// TwinCAT 3 PLC project Test_OnlineChange
// ProgramVersion: 3.1.4026.22
// libraries:
//   Tc2_Standard, * (Beckhoff Automation GmbH)
//   Tc2_System, * (Beckhoff Automation GmbH)
//   Tc3_JsonXml, * (Beckhoff Automation GmbH)
//   Stage, * (_)
// project tree:
//   DUTs/ T_OnlineChangeTestCheck.TcDUT, T_OnlineChangeTestChecks.TcDUT, T_OnlineChangeTestEntity.TcDUT, T_OnlineChangeTestExecute.TcDUT, T_OnlineChangeTestReport.TcDUT, T_OnlineChangeTestRuntime.TcDUT, T_OnlineChangeTestStage.TcDUT, T_OnlineChangeTestWorker.TcDUT
//   GVLs/ GVL_OnlineChangeTest.TcGVL
//   POUs/ FB_OnlineChangeProbe.TcPOU, FB_OnlineChangeDefineReset.TcPOU, FB_OnlineChangeJsonReport.TcPOU, FB_OnlineChangeMovePadding.TcPOU, FB_OnlineChangeStageMarker.TcPOU, FB_FastThreadConfig.TcPOU, FB_TestExecute.TcPOU, FB_TestJob.TcPOU, MAIN.TcPOU
//   / PlcTask.TcTTO
// (motion and I/O tree: see PLC project stage)
// real-time tasks:
//   TASK Example: cycle T#10ms, priority 20, ADS port 350
//   TASK Test: cycle T#10ms, priority 21, ADS port 351
//   TASK VISU_TASK: cycle T#200000us, priority 30, ADS port 352
//   TASK PlcTask: cycle T#10ms, priority 22, ADS port 353
//   TASK PlcTask1: cycle T#10ms, priority 23, ADS port 354
//   TASK PlcTask2: cycle T#10ms, priority 24, ADS port 355

CONFIGURATION Test_OnlineChange
    RESOURCE PLC ON TwinCAT3
        TASK PlcTask(INTERVAL := T#10ms, PRIORITY := 24);
        PROGRAM MAIN WITH PlcTask : MAIN;
    END_RESOURCE
END_CONFIGURATION

// ---- DUTs/T_OnlineChangeTestCheck.TcDUT
TYPE T_OnlineChangeTestCheck :
STRUCT
	bRequired: BOOL;
	bPassed: BOOL;
END_STRUCT
END_TYPE

// ---- DUTs/T_OnlineChangeTestChecks.TcDUT
TYPE T_OnlineChangeTestChecks :
STRUCT
	NoPanic: T_OnlineChangeTestCheck;
	StageSelected: T_OnlineChangeTestCheck;
	StableCallback: T_OnlineChangeTestCheck;
	NoChangeFlags: T_OnlineChangeTestCheck;
	AddDeleteFlags: T_OnlineChangeTestCheck;
	CreatedInit: T_OnlineChangeTestCheck;
	CreatedCallback: T_OnlineChangeTestCheck;
	RepairWarn: T_OnlineChangeTestCheck;
	ActiveJobRunning: T_OnlineChangeTestCheck;
	IdleJobStarted: T_OnlineChangeTestCheck;
	MovedCallback: T_OnlineChangeTestCheck;
	MovedExecuteRunning: T_OnlineChangeTestCheck;
	MovedJobRunning: T_OnlineChangeTestCheck;
END_STRUCT
END_TYPE

// ---- DUTs/T_OnlineChangeTestEntity.TcDUT
TYPE T_OnlineChangeTestEntity :
STRUCT
	nStableInit: UDINT;
	nRemovedInit: UDINT;
	nCreatedInit: UDINT;

	nStableOnlineChange: UDINT;
	bStableLastEntityCreated: BOOL;
	bStableLastEntityDeleted: BOOL;

	nCreatedOnlineChange: UDINT;
	bCreatedLastEntityCreated: BOOL;
	bCreatedLastEntityDeleted: BOOL;

	nMovedInit: UDINT;
	nMovedOnlineChange: UDINT;
	bMovedLastEntityCreated: BOOL;
	bMovedLastEntityDeleted: BOOL;
END_STRUCT
END_TYPE

// ---- DUTs/T_OnlineChangeTestExecute.TcDUT
TYPE T_OnlineChangeTestExecute :
STRUCT
	nMainCycles: UDINT;
	nThreadedCycles: UDINT;
	nMovedCycles: UDINT;
END_STRUCT
END_TYPE

// ---- DUTs/T_OnlineChangeTestReport.TcDUT
TYPE T_OnlineChangeTestReport :
STRUCT
	bAllRequiredPassed: BOOL;
	bRequiredFailure: BOOL;
	bJsonReady: BOOL;
	bJsonCopyOk: BOOL;
	nJsonLength: UDINT;
	sJson: STRING(2048);
END_STRUCT
END_TYPE

// ---- DUTs/T_OnlineChangeTestRuntime.TcDUT
TYPE T_OnlineChangeTestRuntime :
STRUCT
	nMainCycles: UDINT;
	nTotalPanic: UDINT;
	nTotalWarn: UDINT;
END_STRUCT
END_TYPE

// ---- DUTs/T_OnlineChangeTestStage.TcDUT
TYPE T_OnlineChangeTestStage :
STRUCT
	sName: STRING(80);
	nId: UINT;
	iConfiguredFastThread: Stage.I_Thread;
	bFastThreadConfigured: BOOL;
END_STRUCT
END_TYPE

// ---- DUTs/T_OnlineChangeTestWorker.TcDUT
TYPE T_OnlineChangeTestWorker :
STRUCT
	nActiveInit: UDINT;
	nActiveExecute: UDINT;
	nActiveExit: UDINT;
	nIdleInit: UDINT;
	nIdleExecute: UDINT;
	nIdleExit: UDINT;
	nMovedInit: UDINT;
	nMovedExecute: UDINT;
	nMovedExit: UDINT;

	nActiveStartOk: UDINT;
	nActiveStartNone: UDINT;
	nActiveStartError: UDINT;
	nIdleStartOk: UDINT;
	nIdleStartNone: UDINT;
	nIdleStartError: UDINT;
	nMovedStartOk: UDINT;
	nMovedStartNone: UDINT;
	nMovedStartError: UDINT;

	bActiveStartRequested: BOOL;
	bIdleStartRequested: BOOL;
	bMovedStartRequested: BOOL;

	eActiveState: Stage.JobState;
	eIdleState: Stage.JobState;
	eMovedState: Stage.JobState;
END_STRUCT
END_TYPE

// ---- GVLs/GVL_OnlineChangeTest.TcGVL
{attribute 'qualified_only'}
VAR_GLOBAL
	StageState: T_OnlineChangeTestStage;
	Runtime: T_OnlineChangeTestRuntime;
	Entity: T_OnlineChangeTestEntity;
	Execute: T_OnlineChangeTestExecute;
	Worker: T_OnlineChangeTestWorker;
	Checks: T_OnlineChangeTestChecks;
	Report: T_OnlineChangeTestReport;
END_VAR

// ---- POUs/MAIN.TcPOU
// TEST_OC_STAGE values:
// 'INIT' = init baseline
// 'NO_CHANGE' = same-shape online change
// 'REMOVE_THREAD' = remove fast thread
// 'ADD_DELETE_ENTITY' = add/delete entity
// 'MOVE_MEMORY' = force stable instances to move inside program memory
PROGRAM MAIN
{define TEST_OC_STAGE 'MOVE_MEMORY'}
VAR
	fbDefineReset: FB_OnlineChangeDefineReset;
	fbJsonReport: FB_OnlineChangeJsonReport;

	fbStableProbe: FB_OnlineChangeProbe(1);
	fbMainExecute: FB_TestExecute(1);
	fbThreadedExecute: FB_TestExecute(2);
	fbActiveJob: FB_TestJob(1);
	fbIdleJob: FB_TestJob(2);

{IF hasvalue(TEST_OC_STAGE, 'INIT')}
	fbStageInit: FB_OnlineChangeStageMarker(1);
	fbFastThread: Stage.Thread;
	fbFastConfig: FB_FastThreadConfig(fbFastThread);
	fbRemovedProbe: FB_OnlineChangeProbe(2);
{END_IF}
{IF hasvalue(TEST_OC_STAGE, 'NO_CHANGE')}
	fbStageNoChange: FB_OnlineChangeStageMarker(2);
	fbFastThread: Stage.Thread;
	fbFastConfig: FB_FastThreadConfig(fbFastThread);
	fbRemovedProbe: FB_OnlineChangeProbe(2);
{END_IF}
{IF hasvalue(TEST_OC_STAGE, 'REMOVE_THREAD')}
	fbStageRemoveThread: FB_OnlineChangeStageMarker(3);
	fbRemovedProbe: FB_OnlineChangeProbe(2);
{END_IF}
{IF hasvalue(TEST_OC_STAGE, 'ADD_DELETE_ENTITY')}
	fbStageAddDeleteEntity: FB_OnlineChangeStageMarker(4);
	fbCreatedProbe: FB_OnlineChangeProbe(3);
{END_IF}
{IF hasvalue(TEST_OC_STAGE, 'MOVE_MEMORY')}
	fbStageMoveMemory: FB_OnlineChangeStageMarker(5);
	fbFastThread: Stage.Thread;
	fbFastConfig: FB_FastThreadConfig(fbFastThread);
	fbRemovedProbe: FB_OnlineChangeProbe(2);
{END_IF}

{IF hasvalue(TEST_OC_STAGE, 'INIT')}
	fbMovePadInit: FB_OnlineChangeMovePadding;
{END_IF}
{IF hasvalue(TEST_OC_STAGE, 'NO_CHANGE')}
	fbMovePadNoChange: FB_OnlineChangeMovePadding;
{END_IF}
{IF hasvalue(TEST_OC_STAGE, 'REMOVE_THREAD')}
	fbMovePadRemoveThread: FB_OnlineChangeMovePadding;
{END_IF}
{IF hasvalue(TEST_OC_STAGE, 'ADD_DELETE_ENTITY')}
	fbMovePadAddDeleteEntity: FB_OnlineChangeMovePadding;
{END_IF}
{IF hasvalue(TEST_OC_STAGE, 'MOVE_MEMORY')}
	fbMovePadA: FB_OnlineChangeMovePadding;
	fbMovePadB: FB_OnlineChangeMovePadding;
	fbMovePadC: FB_OnlineChangeMovePadding;
{END_IF}

	fbMovedProbe: FB_OnlineChangeProbe(20);
	fbMovedExecute: FB_TestExecute(20);
	fbMovedJob: FB_TestJob(20);
END_VAR

GVL_OnlineChangeTest.Runtime.nMainCycles := GVL_OnlineChangeTest.Runtime.nMainCycles + 1;

IF NOT GVL_OnlineChangeTest.StageState.bFastThreadConfigured THEN
	IF GVL_OnlineChangeTest.StageState.iConfiguredFastThread <> 0 THEN
		fbThreadedExecute.SetThread(GVL_OnlineChangeTest.StageState.iConfiguredFastThread);
		fbActiveJob.SetThread(GVL_OnlineChangeTest.StageState.iConfiguredFastThread);
		fbIdleJob.SetThread(GVL_OnlineChangeTest.StageState.iConfiguredFastThread);
		GVL_OnlineChangeTest.StageState.bFastThreadConfigured := TRUE;
	END_IF
END_IF

Stage.Plant.Run();

IF NOT Stage.Plant.Panicked THEN
	IF NOT GVL_OnlineChangeTest.Worker.bActiveStartRequested THEN
		fbActiveJob.Start();
		GVL_OnlineChangeTest.Worker.bActiveStartRequested := TRUE;
	END_IF

	IF NOT GVL_OnlineChangeTest.Worker.bIdleStartRequested THEN
		IF (GVL_OnlineChangeTest.StageState.nId = 3) OR
			(GVL_OnlineChangeTest.StageState.nId = 4)
		THEN
			fbIdleJob.Start();
			GVL_OnlineChangeTest.Worker.bIdleStartRequested := TRUE;
		END_IF
	END_IF

	IF NOT GVL_OnlineChangeTest.Worker.bMovedStartRequested THEN
		IF GVL_OnlineChangeTest.StageState.nId = 5 THEN
			fbMovedJob.Start();
			GVL_OnlineChangeTest.Worker.bMovedStartRequested := TRUE;
		END_IF
	END_IF
END_IF

GVL_OnlineChangeTest.Worker.eActiveState := fbActiveJob.State;
GVL_OnlineChangeTest.Worker.eIdleState := fbIdleJob.State;
GVL_OnlineChangeTest.Worker.eMovedState := fbMovedJob.State;
GVL_OnlineChangeTest.Runtime.nTotalPanic := Stage.Plant.TotalPanic;
GVL_OnlineChangeTest.Runtime.nTotalWarn := Stage.Plant.TotalWarn;

GVL_OnlineChangeTest.Checks.NoPanic.bRequired := TRUE;
GVL_OnlineChangeTest.Checks.NoPanic.bPassed := GVL_OnlineChangeTest.Runtime.nTotalPanic = 0;

GVL_OnlineChangeTest.Checks.StageSelected.bRequired := TRUE;
GVL_OnlineChangeTest.Checks.StageSelected.bPassed := GVL_OnlineChangeTest.StageState.nId > 0;

GVL_OnlineChangeTest.Checks.StableCallback.bRequired := GVL_OnlineChangeTest.StageState.nId > 1;
GVL_OnlineChangeTest.Checks.StableCallback.bPassed := GVL_OnlineChangeTest.Entity.nStableOnlineChange > 0;

GVL_OnlineChangeTest.Checks.NoChangeFlags.bRequired :=
	(GVL_OnlineChangeTest.StageState.nId = 2) OR
	(GVL_OnlineChangeTest.StageState.nId = 3) OR
	(GVL_OnlineChangeTest.StageState.nId = 5);
GVL_OnlineChangeTest.Checks.NoChangeFlags.bPassed :=
	GVL_OnlineChangeTest.Entity.nStableOnlineChange > 0 AND
	NOT GVL_OnlineChangeTest.Entity.bStableLastEntityCreated AND
	NOT GVL_OnlineChangeTest.Entity.bStableLastEntityDeleted;

GVL_OnlineChangeTest.Checks.AddDeleteFlags.bRequired := GVL_OnlineChangeTest.StageState.nId = 4;
GVL_OnlineChangeTest.Checks.AddDeleteFlags.bPassed :=
	GVL_OnlineChangeTest.Entity.nStableOnlineChange > 0 AND
	GVL_OnlineChangeTest.Entity.bStableLastEntityCreated AND
	GVL_OnlineChangeTest.Entity.bStableLastEntityDeleted;

GVL_OnlineChangeTest.Checks.CreatedInit.bRequired := GVL_OnlineChangeTest.StageState.nId = 4;
GVL_OnlineChangeTest.Checks.CreatedInit.bPassed := GVL_OnlineChangeTest.Entity.nCreatedInit > 0;

GVL_OnlineChangeTest.Checks.CreatedCallback.bRequired := GVL_OnlineChangeTest.StageState.nId = 4;
GVL_OnlineChangeTest.Checks.CreatedCallback.bPassed :=
	GVL_OnlineChangeTest.Entity.nCreatedOnlineChange > 0 AND
	GVL_OnlineChangeTest.Entity.bCreatedLastEntityCreated AND
	GVL_OnlineChangeTest.Entity.bCreatedLastEntityDeleted;

GVL_OnlineChangeTest.Checks.RepairWarn.bRequired := GVL_OnlineChangeTest.StageState.nId = 3;
GVL_OnlineChangeTest.Checks.RepairWarn.bPassed := GVL_OnlineChangeTest.Runtime.nTotalWarn > 0;

GVL_OnlineChangeTest.Checks.ActiveJobRunning.bRequired :=
	(GVL_OnlineChangeTest.StageState.nId = 3) OR
	(GVL_OnlineChangeTest.StageState.nId = 4);
GVL_OnlineChangeTest.Checks.ActiveJobRunning.bPassed := GVL_OnlineChangeTest.Worker.nActiveExecute > 0;

GVL_OnlineChangeTest.Checks.IdleJobStarted.bRequired :=
	(GVL_OnlineChangeTest.StageState.nId = 3) OR
	(GVL_OnlineChangeTest.StageState.nId = 4);
GVL_OnlineChangeTest.Checks.IdleJobStarted.bPassed :=
	GVL_OnlineChangeTest.Worker.nIdleStartOk > 0 AND
	GVL_OnlineChangeTest.Worker.nIdleExecute > 0;

GVL_OnlineChangeTest.Checks.MovedCallback.bRequired := GVL_OnlineChangeTest.StageState.nId = 5;
GVL_OnlineChangeTest.Checks.MovedCallback.bPassed :=
	GVL_OnlineChangeTest.Entity.nMovedOnlineChange > 0 AND
	NOT GVL_OnlineChangeTest.Entity.bMovedLastEntityCreated AND
	NOT GVL_OnlineChangeTest.Entity.bMovedLastEntityDeleted;

GVL_OnlineChangeTest.Checks.MovedExecuteRunning.bRequired := GVL_OnlineChangeTest.StageState.nId = 5;
GVL_OnlineChangeTest.Checks.MovedExecuteRunning.bPassed :=
	GVL_OnlineChangeTest.Execute.nMovedCycles > 0;

GVL_OnlineChangeTest.Checks.MovedJobRunning.bRequired := GVL_OnlineChangeTest.StageState.nId = 5;
GVL_OnlineChangeTest.Checks.MovedJobRunning.bPassed :=
	GVL_OnlineChangeTest.Worker.nMovedStartOk > 0 AND
	GVL_OnlineChangeTest.Worker.nMovedExecute > 0;

GVL_OnlineChangeTest.Report.bAllRequiredPassed :=
	(NOT GVL_OnlineChangeTest.Checks.NoPanic.bRequired OR GVL_OnlineChangeTest.Checks.NoPanic.bPassed) AND
	(NOT GVL_OnlineChangeTest.Checks.StageSelected.bRequired OR GVL_OnlineChangeTest.Checks.StageSelected.bPassed) AND
	(NOT GVL_OnlineChangeTest.Checks.StableCallback.bRequired OR GVL_OnlineChangeTest.Checks.StableCallback.bPassed) AND
	(NOT GVL_OnlineChangeTest.Checks.NoChangeFlags.bRequired OR GVL_OnlineChangeTest.Checks.NoChangeFlags.bPassed) AND
	(NOT GVL_OnlineChangeTest.Checks.AddDeleteFlags.bRequired OR GVL_OnlineChangeTest.Checks.AddDeleteFlags.bPassed) AND
	(NOT GVL_OnlineChangeTest.Checks.CreatedInit.bRequired OR GVL_OnlineChangeTest.Checks.CreatedInit.bPassed) AND
	(NOT GVL_OnlineChangeTest.Checks.CreatedCallback.bRequired OR GVL_OnlineChangeTest.Checks.CreatedCallback.bPassed) AND
	(NOT GVL_OnlineChangeTest.Checks.RepairWarn.bRequired OR GVL_OnlineChangeTest.Checks.RepairWarn.bPassed) AND
	(NOT GVL_OnlineChangeTest.Checks.ActiveJobRunning.bRequired OR GVL_OnlineChangeTest.Checks.ActiveJobRunning.bPassed) AND
	(NOT GVL_OnlineChangeTest.Checks.IdleJobStarted.bRequired OR GVL_OnlineChangeTest.Checks.IdleJobStarted.bPassed) AND
	(NOT GVL_OnlineChangeTest.Checks.MovedCallback.bRequired OR GVL_OnlineChangeTest.Checks.MovedCallback.bPassed) AND
	(NOT GVL_OnlineChangeTest.Checks.MovedExecuteRunning.bRequired OR GVL_OnlineChangeTest.Checks.MovedExecuteRunning.bPassed) AND
	(NOT GVL_OnlineChangeTest.Checks.MovedJobRunning.bRequired OR GVL_OnlineChangeTest.Checks.MovedJobRunning.bPassed);

GVL_OnlineChangeTest.Report.bRequiredFailure :=
	(GVL_OnlineChangeTest.Checks.NoPanic.bRequired AND NOT GVL_OnlineChangeTest.Checks.NoPanic.bPassed) OR
	(GVL_OnlineChangeTest.Checks.StageSelected.bRequired AND NOT GVL_OnlineChangeTest.Checks.StageSelected.bPassed);

GVL_OnlineChangeTest.Report.bJsonReady :=
	GVL_OnlineChangeTest.Report.bAllRequiredPassed OR
	GVL_OnlineChangeTest.Report.bRequiredFailure;

fbJsonReport.Write();

END_PROGRAM

// ---- POUs/FB_OnlineChangeDefineReset.TcPOU
FUNCTION_BLOCK FB_OnlineChangeDefineReset
VAR
END_VAR

METHOD FB_Init : BOOL
VAR_INPUT
	bInitRetains: BOOL;
	bInCopyCode: BOOL;
END_VAR
GVL_OnlineChangeTest.StageState.nId := 0;
GVL_OnlineChangeTest.StageState.sName := 'TEST_OC_UNDEFINED';
GVL_OnlineChangeTest.Report.bJsonReady := FALSE;
GVL_OnlineChangeTest.Report.bJsonCopyOk := FALSE;
GVL_OnlineChangeTest.Report.nJsonLength := 0;
GVL_OnlineChangeTest.Report.sJson := '';
END_METHOD

END_FUNCTION_BLOCK

// ---- POUs/FB_OnlineChangeJsonReport.TcPOU
FUNCTION_BLOCK FB_OnlineChangeJsonReport
VAR
	fbJson: Tc3_JsonXml.FB_JsonSaxPrettyWriter;
END_VAR

METHOD PRIVATE AddCheck
VAR_INPUT
	sName: STRING;
	stCheck: T_OnlineChangeTestCheck;
END_VAR
fbJson.AddKey(sName);
fbJson.StartObject();
fbJson.AddKeyBool('required', stCheck.bRequired);
fbJson.AddKeyBool('passed', stCheck.bPassed);
fbJson.EndObject();
END_METHOD

METHOD Write
VAR_INPUT
END_VAR
fbJson.ResetDocument();
fbJson.StartObject();

fbJson.AddKeyString('stage', GVL_OnlineChangeTest.StageState.sName);
fbJson.AddKeyBool('ready', GVL_OnlineChangeTest.Report.bJsonReady);
fbJson.AddKeyBool('all', GVL_OnlineChangeTest.Report.bAllRequiredPassed);
fbJson.AddKeyBool('fail', GVL_OnlineChangeTest.Report.bRequiredFailure);

fbJson.AddKey('panic');
fbJson.AddUdint(GVL_OnlineChangeTest.Runtime.nTotalPanic);
fbJson.AddKey('warn');
fbJson.AddUdint(GVL_OnlineChangeTest.Runtime.nTotalWarn);

fbJson.AddKey('checks');
fbJson.StartObject();
AddCheck('NoPanic', GVL_OnlineChangeTest.Checks.NoPanic);
AddCheck('StageSelected', GVL_OnlineChangeTest.Checks.StageSelected);
AddCheck('StableCallback', GVL_OnlineChangeTest.Checks.StableCallback);
AddCheck('NoChangeFlags', GVL_OnlineChangeTest.Checks.NoChangeFlags);
AddCheck('AddDeleteFlags', GVL_OnlineChangeTest.Checks.AddDeleteFlags);
AddCheck('CreatedInit', GVL_OnlineChangeTest.Checks.CreatedInit);
AddCheck('CreatedCallback', GVL_OnlineChangeTest.Checks.CreatedCallback);
AddCheck('RepairWarn', GVL_OnlineChangeTest.Checks.RepairWarn);
AddCheck('ActiveJobRunning', GVL_OnlineChangeTest.Checks.ActiveJobRunning);
AddCheck('IdleJobStarted', GVL_OnlineChangeTest.Checks.IdleJobStarted);
AddCheck('MovedCallback', GVL_OnlineChangeTest.Checks.MovedCallback);
AddCheck('MovedExecuteRunning', GVL_OnlineChangeTest.Checks.MovedExecuteRunning);
AddCheck('MovedJobRunning', GVL_OnlineChangeTest.Checks.MovedJobRunning);
fbJson.EndObject();

fbJson.EndObject();

GVL_OnlineChangeTest.Report.nJsonLength := fbJson.CopyDocument(
	GVL_OnlineChangeTest.Report.sJson,
	SIZEOF(GVL_OnlineChangeTest.Report.sJson));
GVL_OnlineChangeTest.Report.bJsonCopyOk := GVL_OnlineChangeTest.Report.nJsonLength > 0;
END_METHOD

END_FUNCTION_BLOCK

// ---- POUs/FB_OnlineChangeProbe.TcPOU
FUNCTION_BLOCK FB_OnlineChangeProbe IMPLEMENTS Stage.I_OnlineChange, Stage.I_Init
VAR
	_ett: Stage.Entity(THIS^);
END_VAR
VAR
	nId: UINT;
END_VAR

METHOD FB_Init : BOOL
VAR_INPUT
	bInitRetains: BOOL;
	bInCopyCode: BOOL;
	nNewId: UINT;
END_VAR
nId := nNewId;
END_METHOD

METHOD Init
VAR_INPUT
END_VAR
CASE nId OF
	1:
		GVL_OnlineChangeTest.Entity.nStableInit := GVL_OnlineChangeTest.Entity.nStableInit + 1;

	2:
		GVL_OnlineChangeTest.Entity.nRemovedInit := GVL_OnlineChangeTest.Entity.nRemovedInit + 1;

	3:
		GVL_OnlineChangeTest.Entity.nCreatedInit := GVL_OnlineChangeTest.Entity.nCreatedInit + 1;

	20:
		GVL_OnlineChangeTest.Entity.nMovedInit := GVL_OnlineChangeTest.Entity.nMovedInit + 1;

END_CASE
END_METHOD

METHOD OnOnlineChange
VAR_INPUT
	bEntityDeleted: BOOL;
	bEntityCreated: BOOL;
END_VAR
CASE nId OF
	1:
		GVL_OnlineChangeTest.Entity.nStableOnlineChange := GVL_OnlineChangeTest.Entity.nStableOnlineChange + 1;
		GVL_OnlineChangeTest.Entity.bStableLastEntityCreated := bEntityCreated;
		GVL_OnlineChangeTest.Entity.bStableLastEntityDeleted := bEntityDeleted;

	3:
		GVL_OnlineChangeTest.Entity.nCreatedOnlineChange := GVL_OnlineChangeTest.Entity.nCreatedOnlineChange + 1;
		GVL_OnlineChangeTest.Entity.bCreatedLastEntityCreated := bEntityCreated;
		GVL_OnlineChangeTest.Entity.bCreatedLastEntityDeleted := bEntityDeleted;

	20:
		GVL_OnlineChangeTest.Entity.nMovedOnlineChange := GVL_OnlineChangeTest.Entity.nMovedOnlineChange + 1;
		GVL_OnlineChangeTest.Entity.bMovedLastEntityCreated := bEntityCreated;
		GVL_OnlineChangeTest.Entity.bMovedLastEntityDeleted := bEntityDeleted;

END_CASE
END_METHOD

METHOD SetId
VAR_INPUT
	nNewId: UINT;
END_VAR
nId := nNewId;
END_METHOD

END_FUNCTION_BLOCK

// ---- POUs/FB_TestExecute.TcPOU
FUNCTION_BLOCK FB_TestExecute IMPLEMENTS Stage.I_Execute
VAR
	_exe: Stage.Execute(THIS^);
END_VAR
VAR
	nId: UINT;
END_VAR

METHOD FB_Init : BOOL
VAR_INPUT
	bInitRetains: BOOL;
	bInCopyCode: BOOL;
	nNewId: UINT;
END_VAR
nId := nNewId;
END_METHOD

METHOD Execute
VAR_INPUT
END_VAR
CASE nId OF
	1:
		GVL_OnlineChangeTest.Execute.nMainCycles := GVL_OnlineChangeTest.Execute.nMainCycles + 1;

	2:
		GVL_OnlineChangeTest.Execute.nThreadedCycles := GVL_OnlineChangeTest.Execute.nThreadedCycles + 1;

	20:
		IF GVL_OnlineChangeTest.StageState.nId = 5 THEN
			GVL_OnlineChangeTest.Execute.nMovedCycles := GVL_OnlineChangeTest.Execute.nMovedCycles + 1;
		END_IF

END_CASE
END_METHOD

METHOD SetThread
VAR_INPUT
	iThread: Stage.I_Thread;
END_VAR
_exe.Thread := iThread;
END_METHOD

METHOD SetId
VAR_INPUT
	nNewId: UINT;
END_VAR
nId := nNewId;
END_METHOD

END_FUNCTION_BLOCK

// ---- POUs/FB_TestJob.TcPOU
FUNCTION_BLOCK FB_TestJob IMPLEMENTS Stage.I_Job
VAR
	_worker: Stage.Worker(THIS^);
END_VAR
VAR
	nId: UINT;
END_VAR

METHOD FB_Init : BOOL
VAR_INPUT
	bInitRetains: BOOL;
	bInCopyCode: BOOL;
	nNewId: UINT;
END_VAR
nId := nNewId;
END_METHOD

METHOD JobExecute
VAR_INPUT
END_VAR
CASE nId OF
	1:
		GVL_OnlineChangeTest.Worker.nActiveExecute := GVL_OnlineChangeTest.Worker.nActiveExecute + 1;

	2:
		GVL_OnlineChangeTest.Worker.nIdleExecute := GVL_OnlineChangeTest.Worker.nIdleExecute + 1;

	20:
		GVL_OnlineChangeTest.Worker.nMovedExecute := GVL_OnlineChangeTest.Worker.nMovedExecute + 1;

END_CASE
END_METHOD

METHOD JobExit
VAR_INPUT
END_VAR
CASE nId OF
	1:
		GVL_OnlineChangeTest.Worker.nActiveExit := GVL_OnlineChangeTest.Worker.nActiveExit + 1;

	2:
		GVL_OnlineChangeTest.Worker.nIdleExit := GVL_OnlineChangeTest.Worker.nIdleExit + 1;

	20:
		GVL_OnlineChangeTest.Worker.nMovedExit := GVL_OnlineChangeTest.Worker.nMovedExit + 1;

END_CASE
END_METHOD

METHOD JobInit
VAR_INPUT
END_VAR
CASE nId OF
	1:
		GVL_OnlineChangeTest.Worker.nActiveInit := GVL_OnlineChangeTest.Worker.nActiveInit + 1;

	2:
		GVL_OnlineChangeTest.Worker.nIdleInit := GVL_OnlineChangeTest.Worker.nIdleInit + 1;

	20:
		GVL_OnlineChangeTest.Worker.nMovedInit := GVL_OnlineChangeTest.Worker.nMovedInit + 1;

END_CASE
END_METHOD

METHOD SetThread
VAR_INPUT
	iThread: Stage.I_Thread;
END_VAR
_worker.Thread := iThread;
END_METHOD

METHOD SetId
VAR_INPUT
	nNewId: UINT;
END_VAR
nId := nNewId;
END_METHOD

METHOD Start : Stage.Result
VAR_INPUT
END_VAR
Start := _worker.Start();

CASE nId OF
	1:
		IF Start > 0 THEN
			GVL_OnlineChangeTest.Worker.nActiveStartOk := GVL_OnlineChangeTest.Worker.nActiveStartOk + 1;
		ELSIF Start = 0 THEN
			GVL_OnlineChangeTest.Worker.nActiveStartNone := GVL_OnlineChangeTest.Worker.nActiveStartNone + 1;
		ELSE
			GVL_OnlineChangeTest.Worker.nActiveStartError := GVL_OnlineChangeTest.Worker.nActiveStartError + 1;
		END_IF

	2:
		IF Start > 0 THEN
			GVL_OnlineChangeTest.Worker.nIdleStartOk := GVL_OnlineChangeTest.Worker.nIdleStartOk + 1;
		ELSIF Start = 0 THEN
			GVL_OnlineChangeTest.Worker.nIdleStartNone := GVL_OnlineChangeTest.Worker.nIdleStartNone + 1;
		ELSE
			GVL_OnlineChangeTest.Worker.nIdleStartError := GVL_OnlineChangeTest.Worker.nIdleStartError + 1;
		END_IF

	20:
		IF Start > 0 THEN
			GVL_OnlineChangeTest.Worker.nMovedStartOk := GVL_OnlineChangeTest.Worker.nMovedStartOk + 1;
		ELSIF Start = 0 THEN
			GVL_OnlineChangeTest.Worker.nMovedStartNone := GVL_OnlineChangeTest.Worker.nMovedStartNone + 1;
		ELSE
			GVL_OnlineChangeTest.Worker.nMovedStartError := GVL_OnlineChangeTest.Worker.nMovedStartError + 1;
		END_IF

END_CASE
END_METHOD

PROPERTY State : Stage.JobState
GET
State := _worker.State;
END_GET
END_PROPERTY

METHOD Stop
VAR_INPUT
END_VAR
_worker.Stop();
END_METHOD

END_FUNCTION_BLOCK

// ---- POUs/FB_OnlineChangeStageMarker.TcPOU
FUNCTION_BLOCK FB_OnlineChangeStageMarker
VAR
END_VAR

METHOD FB_Init : BOOL
VAR_INPUT
	bInitRetains: BOOL;
	bInCopyCode: BOOL;
	nStage: UINT;
END_VAR
GVL_OnlineChangeTest.StageState.nId := nStage;

CASE nStage OF
	1:
		GVL_OnlineChangeTest.StageState.sName := 'TEST_OC_INIT';

	2:
		GVL_OnlineChangeTest.StageState.sName := 'TEST_OC_NO_CHANGE';

	3:
		GVL_OnlineChangeTest.StageState.sName := 'TEST_OC_REMOVE_THREAD';

	4:
		GVL_OnlineChangeTest.StageState.sName := 'TEST_OC_ADD_DELETE_ENTITY';

	5:
		GVL_OnlineChangeTest.StageState.sName := 'TEST_OC_MOVE_MEMORY';

ELSE
	GVL_OnlineChangeTest.StageState.sName := 'TEST_OC_UNDEFINED';

END_CASE
END_METHOD

END_FUNCTION_BLOCK

// ---- POUs/FB_FastThreadConfig.TcPOU
FUNCTION_BLOCK FB_FastThreadConfig
VAR
END_VAR

METHOD FB_Exit : BOOL
VAR_INPUT
	bInCopyCode: BOOL;
END_VAR
IF NOT bInCopyCode THEN
	GVL_OnlineChangeTest.StageState.iConfiguredFastThread := 0;
	GVL_OnlineChangeTest.StageState.bFastThreadConfigured := FALSE;
END_IF
END_METHOD

METHOD FB_Init : BOOL
VAR_INPUT
	bInitRetains: BOOL;
	bInCopyCode: BOOL;
	iThread: Stage.I_Thread;
END_VAR
GVL_OnlineChangeTest.StageState.iConfiguredFastThread := iThread;
END_METHOD

END_FUNCTION_BLOCK

// ---- POUs/FB_OnlineChangeMovePadding.TcPOU
FUNCTION_BLOCK FB_OnlineChangeMovePadding
VAR
	aPadding: ARRAY[1..512] OF UDINT;
END_VAR

END_FUNCTION_BLOCK
